// Input from master arm control task, including arm status and cartesian data
TYPE ST_MasterStatus :
STRUCT
	// master heart beat
	m_masterHeartBeat :INT:=0;
	
	// self-check trigger flag
	m_slaveSelfCheckFlag :BOOL :=FALSE;
	
	// linear motion scale
	m_motionScale : LREAL:=1.5;
	
	// state machine
	m_armState:ARRAY[1..g_mArmNum] OF E_masterArmState;
	
	// index(0 to 4) of slave arm which is tele-linked to master arm
	m_teleSlaveArmIdx :ARRAY[1..g_mArmNum] OF E_MatchedSlaveArmIdx;
	
	// grip angle
	m_gripAngle:ARRAY[1..g_mArmNum] OF LREAL;
	
	// current arm pose in monitor coordinate
	m_curArmPose:ARRAY[1..g_mArmNum] OF ST_Frame;
	
	// current arm twist[linear velocity; angular veloicty] in monitor coordinate
	m_curArmTwist:ARRAY[1..g_mArmNum] OF Vec6d;
	
END_STRUCT
END_TYPE

(* stored: Version 1.1.0.1, ProductVersion 3.1.4024.12
   DUT ST_MasterStatus: Id {3ac2ae6d-6666-445a-980a-7914313359ec} *)
